FUNCTION_BLOCK FB_ReversingSequence
VAR_INPUT
	bEnable 		: BOOL;
	fPosition1 		: LREAL; //pozisyon tiplerimiz LREAL'dir.
	fPosition2 		: LREAL;
	fVelocity		: LREAL;
	tDelay 			: TIME;
END_VAR
VAR_OUTPUT
	bError 			: BOOL;
	sStatus 		: STRING;
END_VAR
VAR
	fbPower			: MC_Power;
	fbMove			: MC_MoveAbsolute;
	nState			: INT;
	fbTimer 		: TON;
END_VAR
VAR_IN_OUT
	Axis		:AXIS_REF;
//Axisler VAR_IN_OUT değişkenleridir sadece onun içinde tanımlanır!!.
END_VAR


fbPower(
	Axis:=Axis , 
	Enable:=TRUE , 
	Enable_Positive:=TRUE, 
	Enable_Negative:=TRUE , 
	Override:=100  );

	fbMove(
	Axis:=Axis , 
	Velocity:=  fVelocity);
	
	Axis.ReadStatus();
	
	fbTimer(PT:= tDelay);
CASE nState OF
	0: //eksenin Enable state'i
		bError 		:=FALSE;
		sStatus 	:='Beklemede';
		IF bEnable AND Axis.Status.Operational THEN
			nState :=10;
			ELSIF NOT Axis.Status.Operational THEN
				nState :=900;
				sStatus :='Enable değil';
		END_IF
		
	10: //Execute state'i
	fbMove.Position :=fPosition1;
	fbMove.Execute := TRUE;
	IF Axis.Status.Moving THEN
		sStatus 	:='1. noktaya Hareket ediyor';
		nState :=20;
		ELSIF Axis.Status.Error OR fbMove.Error THEN
			sStatus 	:='1. noktaya giderken hataya geçti';
			nstate :=900;
	END_IF
	
	20://hareket kontrol state'i
		IF fbMove.Done THEN
			nState := 30;
			fbMove.Execute :=FALSE;
//2. hareketi de yapmak için false dedik.	
			
		END_IF
		
	30:
		
		fbTimer.IN:=TRUE;
		sStatus:='1. Noktada bekliyor.';
		
		IF(fbTimer.Q) THEN
			fbTimer.IN:=FALSE;
			nState:=40;
		END_IF
		
	40://2. hareket.
		fbMove.Position :=fPosition2;
		fbMove.Execute := TRUE;
		IF Axis.Status.Moving THEN
			sStatus 	:='2. noktaya Hareket ediyor';
			nState :=50;
		ELSIF Axis.Status.Error OR fbMove.Error THEN
			sStatus 	:='2. noktaya giderken hataya geçti';
			nstate :=900;
		END_IF
		
	50:
		IF fbMove.Done THEN
			nState := 60;
			fbMove.Execute :=FALSE;
		END_IF
		
	60: 
		fbTimer.IN:=TRUE;
		sStatus:='2. Noktada bekliyor.';
		
		IF(fbTimer.Q) THEN
			fbTimer.IN:=FALSE;
			nState:=0;
		END_IF
		
		
	900:
		bError := TRUE;
		IF NOT bEnable THEN
			fbTimer(IN:=FALSE);
			nState:=0;
		END_IF
		
END_CASE

END_FUNCTION_BLOCK

(* stored: Version 1.1.0.1, ProductVersion 3.1.4024.12
   POU FB_ReversingSequence: Id {c7e436bf-91e9-4e67-87d4-1b1022dd4912}, SpecialFunc None *)
